(* IEC 61131-3 sources: crb-codesys/retrieval/output/codesys_repo/重型运输系统/healthydata/PRG, 3 files *)

(* ---- FileSaver.st ---- *)
PROGRAM FileSaver
VAR
	path 			:STRING:='D:/log';
	intervalMs		:INT := 10;		//间隔时间

	init			:BOOL:= TRUE;
	gi				:INT;
	si				:INT;
	cCtrl			:INT;

	sav				:ARRAY[1..2, 0..10] OF fileSave;
	speed			:INT;
	nowCmd			:ARRAY[1..2, 0..10] OF BOOL;
	canWrite		:ARRAY[1..2, 0..10] OF BOOL;
	nowPosition		:ARRAY[1..2, 0..10] OF INT;
	lastPosition	:ARRAY[1..2, 0..10] OF INT;
	state			:ARRAY[1..2, 0..10] OF INT;
	flag			:ARRAY[1..2, 0..10] OF INT;
END_VAR
VAR CONSTANT
	aOil	:ARRAY [1..7] OF INT :=[9,11,8,8,8,8,23];
END_VAR

//initialize
IF init THEN
	init := FALSE;
	FOR gi := 1 TO 10 DO
		 sav[1, gi](filePath := path, intervalt := intervalMs);
		 sav[1, gi].createDir(gUI.grd[gi].name);
		 init := FALSE;
	END_FOR
	FOR si := 0 TO 10 DO
		 sav[2, si](filePath := path, intervalt := intervalMs);
		 sav[2, si].createDir(gUI.sky[si].name);
		 init := FALSE;
	END_FOR
END_IF

//detect and record ground and sky
FOR gi := 1 TO 10 DO
	 nowCmd[1, gi] := gUI.grd[gi].btnExtend OR gUI.grd[gi].btnRetract;
	 IF nowCmd[1, gi] THEN
		 IF flag[1, gi] = 0 THEN
			 sav[1, gi].new(devName := gUI.grd[gi].name);
			 flag[1, gi] := 1;
		 END_IF
		 //prepare data
		 getGrdData();
		 //write
		 sav[1, gi].write(positionInt := nowPosition[1, gi],speedInt := speed,
			 				 stateInt := state[1, gi]);
	 ELSE
		 IF flag[1, gi] = 1 THEN
			 sav[1, gi].write(positionInt := nowPosition[1, gi],speedInt := speed,
				 				 stateInt := state[1, gi]);
			 sav[1, gi].close();
			 flag[1, gi] := 0;
		 END_IF
	 END_IF
END_FOR

FOR si := 0 TO 10 DO
	 nowCmd[2, si] := gUI.sky[si].btnExtend OR gUI.sky[si].btnRetract;
	 IF nowCmd[2, si] THEN
		 IF flag[2, si] = 0 THEN
			 sav[2, si].new(devName := gUI.sky[si].name);
			 flag[2, si] := 1;
		 END_IF
		 //prepare data
		 getSkyData();
		 //write
		 sav[2, si].write(positionInt := nowPosition[2, si],speedInt := speed,
			 				 stateInt := state[2, si]);
	 ELSE
		 IF flag[2, si] = 1 THEN
			 sav[2, si].write(positionInt := nowPosition[2, si],speedInt := speed,
				 				 stateInt := state[2, si]);
			 sav[2, si].close();
			 flag[2, si] := 0;
		 END_IF
	 END_IF
END_FOR

(* ---- TcpUploader.st ---- *)
PROGRAM TcpUploader
VAR
	destIp 			:STRING:='172.18.150.31';
	destPort 		:UINT:= 61158;
	tcpConnector	:tcpUpload;

	myData 			:ARRAY[1..1024]OF BYTE;
	myDataLen		:__XINT:=21 * 3 + 16;		//总数据长度

	init			:BOOL :=TRUE;
END_VAR

//initialize
IF init THEN
	init := FALSE;
	tcpConnector(InetAddress := destIp,port:= destPort);
END_IF

prepareMetaData();

tcpConnector.send(dataLength := myDataLen, sendBuf := myData);

(* ---- TcpUploader_prepareMetaData_method.st ---- *)
METHOD prepareMetaData
VAR_INPUT
END_VAR
VAR
	gi				:INT;
	si				:INT;

	intTmp			:UINT;
	pos				:INT;
	byte1			:BYTE;
	byte2			:BYTE;
	plugStat		:BYTE;
	destIp 			:STRING:='172.18.150.31';
	destPort 		:UINT:= 61158;
	tcpConnector	:tcpUpload;

	myData 			:ARRAY[1..1024]OF BYTE;
	myDataLen		:__XINT:=21 * 3 + 16;		//总数据长度

	init			:BOOL :=TRUE;
END_VAR

//data head (decimal)
myData[1]	:=	83	;
myData[2]	:=	70	;
myData[3]	:=	68	;
myData[4]	:=	84	;

//data length
myData[5]	:=	0	;
myData[6]	:=	63	;

//healthy data
myData[7]	:=	0	;
myData[8]	:=	11	;

//zero
myData[9]	:=	0	;
myData[10]	:=	0	;
myData[11]	:=	0	;
myData[12]	:=	0	;

myData[13]	:=	0	;
myData[14]	:=	0	;
myData[15]	:=	0	;
myData[16]	:=	0	;

//list
pos := 17;
FOR gi := 1 TO 10 DO
	intTmp := REAL_TO_UINT(gDev.grd[gi].sensor.position * 10);
	byte1 := UINT_TO_BYTE(SHR(intTmp, 8));
	byte2 := UINT_TO_BYTE(intTmp AND 255);
	plugStat := INT_TO_BYTE(gDev.grd[gi].state);

	myData[pos] := plugStat;
	pos := pos + 1;
	myData[pos] := byte1;
	pos := pos + 1;
	myData[pos] := byte2;
	pos := pos + 1;
END_FOR
FOR si := 0 TO 10 DO
	intTmp := REAL_TO_UINT(gDev.sky[si].sensor.position * 10);
	byte1 := UINT_TO_BYTE(SHR(intTmp, 8));
	byte2 := UINT_TO_BYTE(intTmp AND 255);
	plugStat := INT_TO_BYTE(gDev.sky[si].state);

	myData[pos] := plugStat;
	pos := pos + 1;
	myData[pos] := byte1;
	pos := pos + 1;
	myData[pos] := byte2;
	pos := pos + 1;
END_FOR
